// TIA Portal V19 export
FUNCTION_BLOCK "SinamicsCU"   // FB129, LAD
TITLE = Sinamics CU
// stored: Access Published, MemoryReserve 100, SetENOAutomatically false
   VAR_INPUT
      Rst : Bool;   // Reset alarms
      Tel393_HWID : HW_IO;   // Telegram 370 for path test and diagnostic
      AccessPoint : HW_IO;   // AccessPoint for SinaParaS
      AxisID : USInt;   // Axis ID for SinaParaS
      TokenChain : Int;   // Number of token chain for SinaParaS
      Simulation : Bool;
   END_VAR
   VAR_OUTPUT
      AlarmPresence : Bool;   // Cumulative alarm presence
      WarningPresence : Bool;   // Cumulative warning presence
   END_VAR
   VAR_IN_OUT
      Alarm : "SinamicsCU_Alarms";
      Warning : "SinamicsCU_Warnings";
      Diag : "TO_Diagnostic";
   END_VAR
   VAR
      GetTelIn : GETIO;
      SetTelOut : SETIO_PART;
      ReadAlarm : "RW_SINAMICS_Par";
      ReadWarning : "RW_SINAMICS_Par";
      PathTest : Array[1..4] of "PathTestSignal";
   END_VAR
   VAR_TEMP
      TEL_IN : "Tel393In_PM";
      TEL_OUT : "Tel393Out_PM";
   END_VAR
BEGIN

REGION Network 1 (SCL): Info
   //=============================================================================
   //PM FORMING
   //-----------------------------------------------------------------------------
   // Library: StandardBlocks
   // Tested with: S7-1518TF
   // Engineering: TIA Portal V18
   // Restrictions: -
   // Requirements: S7-1500
   // Functionality: Sinamics CU device
   //
   // v1.0.0  28/12/2022 
   // v1.1.0  14/02/2022 Simulation added
   //=============================================================================
END_REGION

REGION Network 2: Read data from CU / Read consistent data of an IO (sub)module
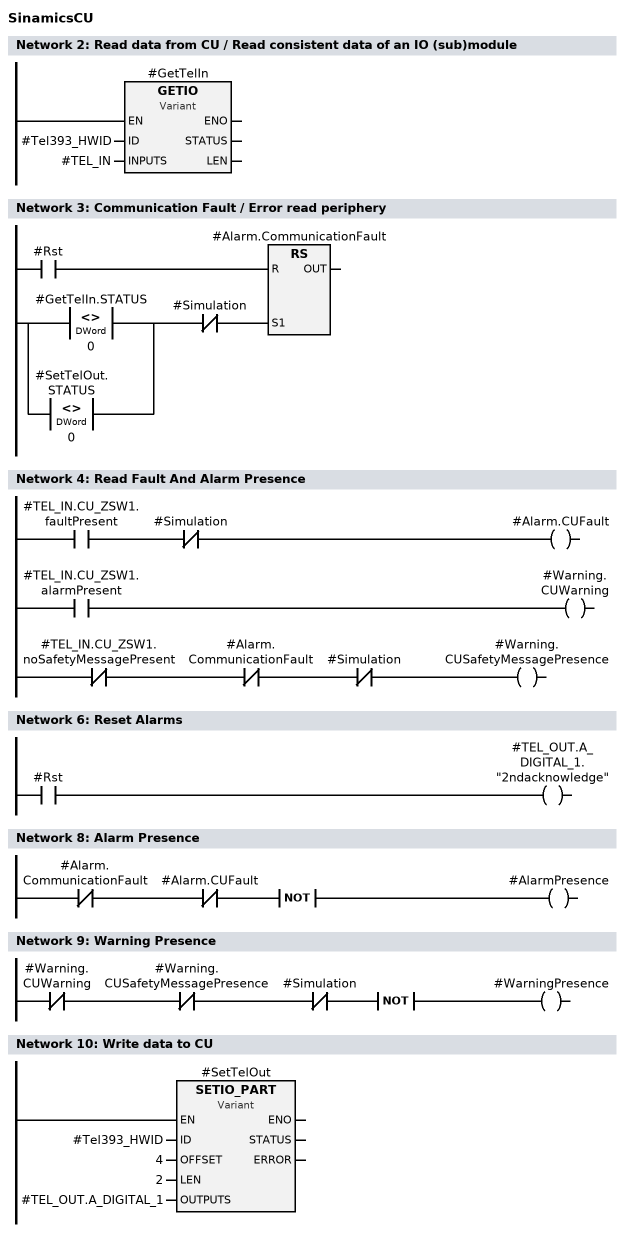
   RUNG wire#powerrail
      { S7_Templates := "[ptr_type := Variant, id_type := HW_SUBMODULE]" } #GetTelIn.GETIO(ID := #Tel393_HWID, INPUTS := #TEL_IN, STATUS =>, LEN =>)
   END_RUNG
   // the same network as SCL:
   #GetTelIn(ID := #Tel393_HWID, INPUTS := #TEL_IN);   // GETIO
END_REGION

REGION Network 3: Communication Fault / Error read periphery
   RUNG wire#powerrail
      Contact( #Rst )
      S_RS(operand := #Alarm.CommunicationFault, s1 := wire#w2)
   END_RUNG
   RUNG wire#powerrail
      { S7_Templates := "SrcType := DWord" } NE_Contact(in1 := #GetTelIn.STATUS, in2 := 0)
      wire#w1
      I_Contact( #Simulation )
   END_RUNG wire#w2
   RUNG wire#powerrail
      { S7_Templates := "SrcType := DWord" } NE_Contact(in1 := #SetTelOut.STATUS, in2 := 0)
   END_RUNG wire#w1
   // the same network as SCL:
   IF #Rst THEN
       #Alarm.CommunicationFault := FALSE;   // RS flip-flop
   END_IF;
   IF ((#GetTelIn.STATUS <> 0) OR (#SetTelOut.STATUS <> 0)) AND NOT #Simulation THEN
       #Alarm.CommunicationFault := TRUE;
   END_IF;
END_REGION

REGION Network 4: Read Fault And Alarm Presence
   RUNG wire#powerrail
      Contact( #TEL_IN.CU_ZSW1.faultPresent )
      I_Contact( #Simulation )
      Coil( #Alarm.CUFault )
   END_RUNG
   RUNG wire#powerrail
      Contact( #TEL_IN.CU_ZSW1.alarmPresent )
      Coil( #Warning.CUWarning )
   END_RUNG
   RUNG wire#powerrail
      I_Contact( #TEL_IN.CU_ZSW1.noSafetyMessagePresent )
      I_Contact( #Alarm.CommunicationFault )
      I_Contact( #Simulation )
      Coil( #Warning.CUSafetyMessagePresence )
   END_RUNG
   // the same network as SCL:
   #Alarm.CUFault := #TEL_IN.CU_ZSW1.faultPresent AND NOT #Simulation;
   #Warning.CUWarning := #TEL_IN.CU_ZSW1.alarmPresent;
   #Warning.CUSafetyMessagePresence := NOT #TEL_IN.CU_ZSW1.noSafetyMessagePresent AND NOT #Alarm.CommunicationFault AND NOT #Simulation;
END_REGION

REGION Network 5 (SCL): Diganostic

   #Diag.DeviceType := 1;
   #Diag.TO_SimulationActive := #Simulation;

   IF #AccessPoint > 0 AND #TokenChain > 0 AND NOT #Simulation THEN

       #ReadAlarm(Enable := #Alarm.CUFault,
                  ReadWrite := 0,
                  ParNo := 2131,
                  Index := 0,
                  AxisNo := #AxisID,
                  HW_ID := #AccessPoint,
                  TokenChain := #TokenChain);

       #ReadWarning(Enable := #Warning.CUWarning AND NOT #Alarm.CUFault,
                    ReadWrite := 0,
                    ParNo := 2132,
                    Index := 0,
                    AxisNo := #AxisID,
                    HW_ID := #AccessPoint,
                    TokenChain := #TokenChain);


       IF #Alarm.CUFault THEN
           IF #ReadAlarm.Done THEN
               #Diag.Drive_Message := REAL_TO_UINT(#ReadAlarm.ValueReadReal);
           END_IF;
       ELSIF #Warning.CUWarning THEN
           IF #ReadWarning.Done THEN
               #Diag.Drive_Message := REAL_TO_UINT(#ReadWarning.ValueReadReal);
           END_IF;
       ELSE
           #Diag.Drive_Message := 0;
       END_IF;

       #Diag.Drive_ErrorPresence := #Alarm.CUFault;
   ELSE
       #Diag.Drive_Message := 0;
       #Diag.Drive_ErrorPresence := FALSE;
   END_IF;

   IF #AlarmPresence THEN
       #Diag.MessageType := 2;
   ELSIF #WarningPresence THEN
       #Diag.MessageType := 1;
   ELSE
       #Diag.MessageType := 0;
   END_IF;
END_REGION

REGION Network 6: Reset Alarms
   RUNG wire#powerrail
      Contact( #Rst )
      Coil( #TEL_OUT.A_DIGITAL_1."2ndacknowledge" )
   END_RUNG
   // the same network as SCL:
   #TEL_OUT.A_DIGITAL_1."2ndacknowledge" := #Rst;
END_REGION

REGION Network 7 (SCL): Path test
   //Read path test Info 
   #PathTest[1].TestRequired := #TEL_IN.E_DIGITAL_1.Axis1_PathTestReq;
   #PathTest[1].TestRunning := #TEL_IN.E_DIGITAL_1.Axis1_PathTestRunning;
   #PathTest[2].TestRequired := #TEL_IN.E_DIGITAL_1.Axis2_PathTestReq;
   #PathTest[2].TestRunning := #TEL_IN.E_DIGITAL_1.Axis2_PathTestRunning;
   #PathTest[3].TestRequired := #TEL_IN.E_DIGITAL_1.Axis3_PathTestReq;
   #PathTest[3].TestRunning := #TEL_IN.E_DIGITAL_1.Axis3_PathTestRunning;
   #PathTest[4].TestRequired := #TEL_IN.E_DIGITAL_1.Axis4_PathTestReq;
   #PathTest[4].TestRunning := #TEL_IN.E_DIGITAL_1.Axis4_PathTestRunning;


   //Write Path Test out
   #TEL_OUT.A_DIGITAL_1.PathTestAxis1 := #PathTest[1].TestRunCmd;
   #TEL_OUT.A_DIGITAL_1.PathTestAxis2 := #PathTest[2].TestRunCmd;
   #TEL_OUT.A_DIGITAL_1.PathTestAxis3 := #PathTest[3].TestRunCmd;
   #TEL_OUT.A_DIGITAL_1.PathTestAxis4 := #PathTest[4].TestRunCmd;
END_REGION

REGION Network 8: Alarm Presence
   RUNG wire#powerrail
      I_Contact( #Alarm.CommunicationFault )
      I_Contact( #Alarm.CUFault )
      Not()
      Coil( #AlarmPresence )
   END_RUNG
   // the same network as SCL:
   #AlarmPresence := NOT (NOT #Alarm.CommunicationFault AND NOT #Alarm.CUFault);
END_REGION

REGION Network 9: Warning Presence
   RUNG wire#powerrail
      I_Contact( #Warning.CUWarning )
      I_Contact( #Warning.CUSafetyMessagePresence )
      I_Contact( #Simulation )
      Not()
      Coil( #WarningPresence )
   END_RUNG
   // the same network as SCL:
   #WarningPresence := NOT (NOT #Warning.CUWarning AND NOT #Warning.CUSafetyMessagePresence AND NOT #Simulation);
END_REGION

REGION Network 10: Write data to CU
   RUNG wire#powerrail
      { S7_Templates := "[ptr_type := Variant, id_type := HW_SUBMODULE]" } #SetTelOut.SETIO_PART(ID := #Tel393_HWID, OFFSET := 4, LEN := 2, OUTPUTS := #TEL_OUT.A_DIGITAL_1, STATUS =>, ERROR =>)
   END_RUNG
   // the same network as SCL:
   #SetTelOut(ID := #Tel393_HWID, OFFSET := 4, LEN := 2, OUTPUTS := #TEL_OUT.A_DIGITAL_1);   // SETIO_PART
END_REGION
END_FUNCTION_BLOCK
